(* IEC 61131-3 sources: plc-release/libs, 13 files *)

(* ---- CMP.st ---- *)
FUNCTION_BLOCK CMP
VAR_INPUT
IN1 : DINT := 0 ;
IN2 : DINT := 0 ;
END_VAR

VAR_OUTPUT
LT : BOOL := FALSE ;
EQ : BOOL := FALSE ;
QT : BOOL := FALSE ;
END_VAR

IF  ( IN1 < IN2 )  THEN
LT := TRUE ;
END_IF ;
IF  ( IN1 = IN2 )  THEN
EQ := TRUE ;
END_IF ;
IF  ( IN1 > IN2 )  THEN
QT := TRUE ;
END_IF ;

END_FUNCTION_BLOCK

(* ---- CONNECT.st ---- *)
FUNCTION_BLOCK CONNECT
VAR_INPUT
ENC : BOOL;
PARTNER : STRING;
END_VAR

VAR_OUTPUT
VALID : BOOL := FALSE ;
ERROR : BOOL := FALSE ;
STATUS : DINT := 0 ;
ID : STRING := "";
END_VAR

VAR
TEMP : BOOL := FALSE ;
END_VAR

  IF ENC = TRUE THEN
    TEMP := connectRequest(PARTNER);
  END_IF ;

  IF VALID = TRUE AND ENC = FALSE THEN
    TEMP := disconnect(PARTNER);
  END_IF ;

  IF isConnected(PARTNER) THEN
    VALID := TRUE ;
    ERROR := FALSE ;
    STATUS := 0;
    ID := PARTNER ;
  ELSE
    VALID := FALSE ;
    ERROR := TRUE ;
    STATUS := 1;
  END_IF ;

END_FUNCTION_BLOCK

(* ---- CTD.st ---- *)
FUNCTION_BLOCK CTD
VAR_INPUT
  CD : BOOL := FALSE  ;
  LD : BOOL := FALSE ;
  PV : DINT :=  0 ;
END_VAR

VAR_OUTPUT
Q : BOOL := FALSE ;
CV : DINT :=  0 ;
END_VAR

IF LD THEN CV := PV ;
ELSIF CD AND (CV > PV)
THEN CV := CV - 1 ;
END_IF ;

Q := (CV <= 0) ;

END_FUNCTION_BLOCK

(* ---- CTU.st ---- *)
FUNCTION_BLOCK CTU
VAR_INPUT
CU : BOOL := FALSE ;
R : BOOL := FALSE ;
PV : DINT := 0 ;
END_VAR

VAR_OUTPUT
Q : BOOL := FALSE  ;
CV : DINT :=  0 ;
END_VAR

IF R THEN CV := 0 ;
ELSIF CU AND ( CV < PV )
THEN CV := CV + 1;
END_IF ;

Q := (CV >= PV) ;

END_FUNCTION_BLOCK

(* ---- CTUD.st ---- *)
FUNCTION_BLOCK CTUD

VAR_INPUT
CU : BOOL := FALSE  ;
CD : BOOL := FALSE  ;
R : BOOL := FALSE  ;
LD : BOOL := FALSE  ;
PV : DINT :=  0  ;
END_VAR

VAR_OUTPUT
QU : BOOL := FALSE  ;
QD : BOOL := FALSE ;
CV : DINT :=  0  ;
END_VAR

IF R THEN CV := 0 ;
ELSIF LD THEN CV := PV ;
ELSE
    IF NOT (CU AND CD) THEN
        IF CU AND (CV < PV)
        THEN CV := CV + 1 ;
        ELSIF CD AND (CV > PV)
        THEN CV := CV - 1 ;
        END_IF ;
    END_IF ;
END_IF ;
QU := (CV >= PV) ;
QD := (CV <= 0) ;

END_FUNCTION_BLOCK

(* ---- F_TRIG.st ---- *)
FUNCTION_BLOCK F_TRIG
VAR
M : BOOL := FALSE ;
END_VAR

VAR_INPUT
CLK : BOOL := FALSE ;
END_VAR

VAR_OUTPUT
Q : BOOL := FALSE ;
END_VAR

Q := NOT CLK AND NOT M;
M := NOT CLK ;

END_FUNCTION_BLOCK

(* ---- PLS.st ---- *)
FUNCTION_BLOCK PLS
VAR
PEROID_CHECKER : TIME := 0  ;
FIRST_CHECKER : BOOL := TRUE;
END_VAR

VAR_INPUT
RUN : BOOL := FALSE ;
CYCLE : TIME :=  0 ;
END_VAR

VAR_OUTPUT
Q : BOOL := FALSE ;
END_VAR

IF (FIRST_CHECKER) THEN
  FIRST_CHECKER := FALSE ;
  PEROID_CHECKER  := @#timerValue ;
END_IF ;

IF (RUN AND (@#timerValue  - PEROID_CHECKER ) >= CYCLE) THEN
  PEROID_CHECKER := @#timerValue ;
END_IF ;

IF (RUN AND (@#timerValue - PEROID_CHECKER ) >= (CYCLE - @#cycleValue) ) THEN
  Q := TRUE ;
END_IF ;

IF (NOT RUN ) THEN
  Q := FALSE ;
END_IF ;

END_FUNCTION_BLOCK

(* ---- R_TRIG.st ---- *)
FUNCTION_BLOCK R_TRIG
VAR
M : BOOL := FALSE ;
END_VAR

VAR_INPUT
CLK : BOOL := FALSE  ;
END_VAR

VAR_OUTPUT
Q : BOOL := FALSE  ;
END_VAR

Q := CLK AND NOT M ;
M := CLK ;

END_FUNCTION_BLOCK

(* ---- TON.st ---- *)
FUNCTION_BLOCK TON
VAR_INPUT
IN : BOOL := FALSE ;
PT : TIME := 0 ;
END_VAR

VAR_OUTPUT
Q : BOOL := FALSE ;
ET : TIME := 0 ;
END_VAR

VAR
H : BOOL := FALSE ;
END_VAR

  IF NOT IN OR NOT H THEN
    Q  :=  FALSE ;
    ET  :=  T# 0 ms ;
    @#timerSetValue(T# 0 ms) ;
  ELSE
     IF @#timerValue >= PT THEN
      ET  :=  PT ;
      Q  :=  TRUE ;
      ELSE
      ET  :=  @#timerValue ;
    END_IF ;
  END_IF ;

  H := IN ;

END_FUNCTION_BLOCK

(* ---- TP.st ---- *)
FUNCTION_BLOCK TP
VAR_INPUT
IN : BOOL := FALSE ;
PT : TIME := 0 ;
END_VAR

VAR_OUTPUT
Q : BOOL := FALSE  ;
ET : TIME := 0  ;
END_VAR

  IF (NOT IN AND NOT Q) THEN
    Q := FALSE ;
    ET := T# 0 ms ;
    @#timerSetValue(T# 0 ms) ;
  END_IF ;

  IF IN  THEN
    Q := TRUE ;
    ET := @#timerValue ;
  END_IF ;

  IF (@#timerValue >= PT ) THEN
    ET := PT ;
    Q := FALSE ;
    END_IF ;

END_FUNCTION_BLOCK

(* ---- URCV.st ---- *)
FUNCTION_BLOCK URCV
VAR_INPUT
ENR : BOOL;
ID : STRING := "";
RID : STRING := "";
END_VAR

VAR_OUTPUT
NDR : BOOL := FALSE ;
ERROR : BOOL := FALSE ;
STATUS : DINT := 0 ;
DATA : ANY := 0;
END_VAR

VAR
THIS : STRING ;
RESULT : ANY ;
END_VAR

  IF NDR THEN
    NDR := FALSE ;
    ERROR := FALSE ;
    STATUS := 0 ;
  END_IF ;

  IF isConnected(ID) = FALSE THEN
    ERROR := TRUE ;
    STATUS := 1 ;
    RETURN ;
  END_IF ;

  THIS := thisBlock ;
  RESULT := rcvData(ID, RID, THIS) ;

  IF RESULT <> rcvError THEN
    NDR := TRUE ;
    ERROR := FALSE ;
    STATUS := 0 ;
    DATA := RESULT ;
  ELSE
    NDR := FALSE ;
    ERROR := TRUE ;
    STATUS := 1 ;
  END_IF ;

END_FUNCTION_BLOCK

(* ---- USEND.st ---- *)
FUNCTION_BLOCK USEND
VAR_INPUT
REQ : BOOL;
COMMCHANNEL : STRING := "";
RID : STRING := "";
DATA : ANY := 0;
END_VAR

VAR_OUTPUT
DONE : BOOL := FALSE ;
ERROR : BOOL := FALSE ;
STATUS : DINT := 0 ;
END_VAR

VAR
THIS : STRING ;
RESULT : BOOL := FALSE ;
END_VAR

  IF RESULT THEN
    DONE := FALSE ;
    ERROR := FALSE ;
    STATUS := 0 ;
  END_IF ;

  IF isConnected(COMMCHANNEL) = FALSE THEN
    DONE := FALSE ;
    ERROR := TRUE ;
    STATUS := 1 ;
  END_IF ;

  THIS := thisBlock ;
  RESULT := sendData(COMMCHANNEL, THIS, RID, DATA) ;

  IF RESULT THEN
    DONE := TRUE ;
    ERROR := FALSE ;
    STATUS := 0 ;
  END_IF ;

END_FUNCTION_BLOCK

(* ---- WRCV.st ---- *)
FUNCTION_BLOCK URCV
VAR_INPUT
ENR : BOOL;
ID : STRING := "";
RID : STRING := "";
END_VAR

VAR_OUTPUT
NDR : BOOL := FALSE ;
ERROR : BOOL := FALSE ;
STATUS : DINT := 0 ;
DATA : ANY := 0;
END_VAR

VAR
THIS : STRING ;
RESULT : ANY ;
END_VAR

  IF NDR THEN
    NDR := FALSE ;
    ERROR := FALSE ;
    STATUS := 0 ;
  END_IF ;

  IF isConnected(ID) = FALSE THEN
    ERROR := TRUE ;
    STATUS := 1 ;
    RETURN ;
  END_IF ;

  THIS := thisBlock ;
  RESULT := wrcvData(ID, RID, THIS) ;

  IF RESULT <> rcvError THEN
    NDR := TRUE ;
    ERROR := FALSE ;
    STATUS := 0 ;
    DATA := RESULT ;
  ELSE
    NDR := FALSE ;
    ERROR := TRUE ;
    STATUS := 1 ;
  END_IF ;

END_FUNCTION_BLOCK
